// TIA Portal project "Switch and Timer Output Logic" (V17)
// PLC Example 32
// When Switch is turned ON, Output 1 and Output 2 will be ON.
// When Switch is turned OFF, Output 1 will be OFF after 10 sec and Output 2 will be OFF after 15 sec.

(* hardware
DEVICE "S7-1200 station_1"  S7-1200 Station
   slot 0: "Rack_0"  S7-1200 Rack  Rack  V1.0
   slot 1: "PLC_1"  CPU 1212C DC/DC/Rly  6ES7 212-1HE40-0XB0  V4.5
*)

// ===== PLC "PLC_1"  CPU 1212C DC/DC/Rly =====

VAR_GLOBAL   // PLC tag table "Default tag table"
   "Switch_On" AT %I0.0 : Bool;
   "Switch_Off" AT %I0.1 : Bool;
   "Valve1" AT %Q0.0 : Bool;
   "Valve2" AT %Q0.1 : Bool;
   "Tag_1" AT %M0.0 : Bool;
END_VAR

// folder: System blocks/Program resources

DATA_BLOCK "IEC_Timer_0_DB"   // DB1
{ S7_Optimized_Access := 'TRUE' }
AUTHOR : Simatic
FAMILY : IEC
NAME : IEC_TMR
VERSION : 1.0
// stored: InstanceOfName IEC_TIMER
"IEC_TIMER"
BEGIN
END_DATA_BLOCK

DATA_BLOCK "IEC_Timer_0_DB_1"   // DB2
{ S7_Optimized_Access := 'TRUE' }
AUTHOR : Simatic
FAMILY : IEC
NAME : IEC_TMR
VERSION : 1.0
// stored: InstanceOfName IEC_TIMER
"IEC_TIMER"
BEGIN
END_DATA_BLOCK

// folder: (top level)

ORGANIZATION_BLOCK "Main"   // OB1, LAD, ProgramCycle
TITLE = "Main Program Sweep (Cycle)"
{ S7_Optimized_Access := 'TRUE' }
VERSION : 0.1
   VAR_INPUT
      Initial_Call : Bool;   // Initial call of this OB
      Remanence : Bool;   // =True, if remanent data are available
   END_VAR
BEGIN

REGION Network 1
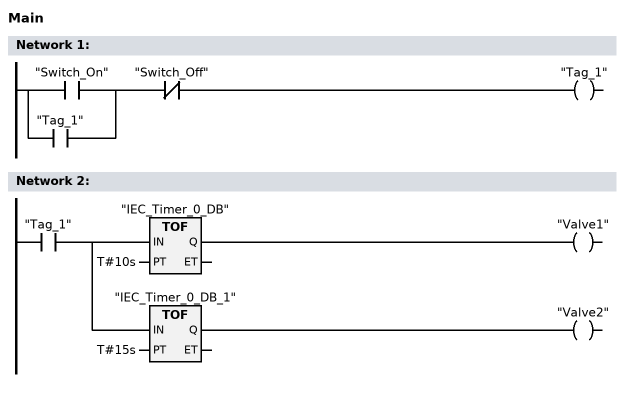
   RUNG wire#powerrail
      Contact( "Switch_On" )
      wire#w1
      I_Contact( "Switch_Off" )
      Coil( "Tag_1" )
   END_RUNG
   RUNG wire#powerrail
      Contact( "Tag_1" )
   END_RUNG wire#w1
   // the same network as SCL:
   "Tag_1" := ("Switch_On" OR "Tag_1") AND NOT "Switch_Off";
END_REGION

REGION Network 2
   "IEC_Timer_0_DB".TOF(IN := "Tag_1", PT := T#10s);
   "Valve1" := "IEC_Timer_0_DB".Q;
   "IEC_Timer_0_DB_1".TOF(IN := "Tag_1", PT := T#15s);
   "Valve2" := "IEC_Timer_0_DB_1".Q;
END_REGION
END_ORGANIZATION_BLOCK